TYPE ST_SampleSlot :
(*
    Represents a general slot for a sample puck.
*)
STRUCT
    {attribute 'pytmc' := '
        pv: eState
        io: io
        field: DESC Enumeration of possible states for a slot in the sample delivery system. (empty, full, or disabled)
    '}
    eState: E_SampleSlotStates;
    {attribute 'pytmc' := '
        pv: sTag
        io: i
        field: DESC A two character identifier for the slot. e.g., T1, B3, etc...
    '}
    sTag: STRING;
    {attribute 'pytmc' := '
        pv: sDesc
        io: io
        field: DESC If the slot is in the full state, this value is supposed to describe what is in the slot.
    '}
    sDesc: STRING;
END_STRUCT
END_TYPE

(* stored: Version 1.1.0.1
   DUT ST_SampleSlot: Id {09c3dd66-8f5a-4524-bfed-dea9564f5621} *)
